# EPICS autosave request: asApp/Db/configMenu.req
$(P)$(CONFIG)Menu:currName
$(P)$(CONFIG)Menu:currDesc
